DATA_BLOCK "DB_PLT_Non_Trk_Tmp_T_this_is_a_pretty_long_title"
TITLE = %version: 5.10 % %Commit:  fbddf08d % CN: 20
{ S7_Optimized_Access := 'FALSE' }
FAMILY : Tubtrax
VERSION : 0.0
//
//SOURCE
//%Project:      allcttt %
//%Repo:         a_ttt %
//%Commit:       fbddf08d %
//%DateTimeUTC:  2024-05-14T09:13:31 %
//
//%HISTORY%
//Issue:        Commit:  Date:      Version: Author:              Description:
//------------- -------- ---------- -------- -------------------- ------------------------------------------------------------------------------
//ALLCTTT-4214  fbddf08d 2024-05-14 5.10     Henri de Leijer      disable_receive plt interface to lib
//ALLCTTT-4059  c3808b61 2023-12-11 5.09     Pascal van Kempen    Added history table
//ALLCTTT-4042  a864e0dd 2023-12-06 5.08     Harm Hopmans         Renamed folders that contained space character
//ALLCTTT-4042  55fd833f 2023-12-05 5.07     Henri de Leijer      First step to remove the library files
//ALLCTTT-272   544e4e84 2020-12-10 5.06     Pascal van Kempen    removed keywords
//ALLCTTT-272   9d531fbf 2020-12-10 5.05     Pascal van Kempen    Revert corrected checkin sequence for determining version information properly
//ALLCTTT-272   ae3fa862 2020-12-10 5.04     Pascal van Kempen    corrected checkin sequence for determining version information properly
//ALLCTTT-272   5a1edb78 2020-12-10 5.03     Pascal van Kempen    Revert keywords updates
//ALLCTTT-272   8d62c219 2020-12-10 5.02     Pascal van Kempen    keywords updates
//ALLCTTT-272   31a64871 2020-12-10 5.01     Pascal van Kempen    initial import
//
//Modification History:                                 By:      Date:     Rev:
//----------------------------------------------------  -------  --------  -----
//ra#31964: Based on 2.15.0.0 version 1.02              nlhhop   14-01-19   2.01
   STRUCT
      Entries_Used : Int;   // Number of entries used in tracking DB
      Displacement : Int;   // Displacement last PLC cycle used by read tracking functions
      Entries_Present : Int;   // Number of entries present in tracking DB
      DB_PLT_nr_Upstream : Int;   // DB PLT number of the upstream
      DB_PLT_nr_Downstream : Int;   // DB PLT number of the downstream
      Done : Bool;   // Header data is written in the PLT DB.
      Motor_Run : Bool;   // Motor running signal
      Motor_On_Speed : Bool;   // Motor on speed signal
      Cascade_Start_up : Bool;   // Cascade start up downstream
      Section_Available : Bool;   // Section is available to recieve items (TEP=1)
      Section_Operational : Bool;   // Section is started
      Item_at_Handover : Bool;   // Item at Handover position
      PEC_Latch : Bool;   // PEC Latch at EOS
      Inhibit_Receive_Item : Bool;   // Section is setting the inhibit to receive item found in upstream handover
      Section_Stopped : Bool;   // Section is stopped. (Actuele speed = 0)
      Disable_Receive : Bool;   // Section is disabled to receive items
      Length_Section : Int;   // Length of the conveyor
      Entry : Array[1..300] of "UDT_PLT_Entry";
   END_STRUCT;


BEGIN

END_DATA_BLOCK
